(*			
	EVERDE sp. z o.o.
	Rafał Osajda		22.01.2025		TC 4026.13		wer. 0.0.0.1
	B_Baza dla czujników binarnych styk normalnie zamkniety 	
*)
FUNCTION_BLOCK FB_Sensor_NC EXTENDS FB_Sensor
VAR
END_VAR

METHOD FB_init : BOOL
VAR_INPUT
	bInitRetains : BOOL; // if TRUE, the retain variables are initialized (warm start / cold start)
	bInCopyCode : BOOL;  // if TRUE, the instance afterwards gets moved into the copy code (online change)
END_VAR
THIS^.eType		:= E_SensorType.NC;
END_METHOD

(*			
	EVERDE sp. z o.o.
	Rafał Osajda		05.02.2025		TC 4026.13		wer. 0.0.0.1
	Zwraca aktualny stan czujnika
*)
METHOD IsActive : BOOL
IsActive				:= NOT THIS^.bContact;
END_METHOD

END_FUNCTION_BLOCK

(* stored: Version 1.1.0.1
   POU FB_Sensor_NC: Id {66f34a47-e680-4956-881b-083b97d3eeed}, SpecialFunc None
   Method FB_init: Id {834e05af-13c9-4454-a99d-74f1de00ecd0}
   Method IsActive: Id {f7918a5a-9f4d-4c0c-9ba4-df583fdafefe} *)
